PROGRAM OverridePressure
VAR
	fb_SetPressure : FB_SetChamberPressure;
END_VAR

fb_SetPressure(chamber := st_GMD, rNewPressure := New_Pressure, Override := Global_OverridePressure);

END_PROGRAM

(* stored: Version 1.1.0.1, ProductVersion 3.1.4022.12
   POU OverridePressure: Id {5b50903e-4143-408a-8dab-1e1782813793}, SpecialFunc None *)
